//==================================================================================================
//								RJM Maszyny sp. z o.o.
//									13.05.2022
//
//	Obsługa przycisku niepodświetlanego
//	v1.0	|| TC v 3.1.4024.22		|| - pierwsza wersja
//==================================================================================================
INTERFACE I_Przycisk

//==================================================================================================
//								RJM Maszyny sp. z o.o.
//									13.05.2022
//
//	Sprawdzenie czy wciśnięty
//	v1.0	|| TC v 3.1.4024.22		|| - pierwsza wersja
//==================================================================================================
PROPERTY CzyNacisniety : Bool
GET
END_GET
END_PROPERTY

//==================================================================================================
//								RJM Maszyny sp. z o.o.
//									13.05.2022
//
//	Sprawdzenie czy puszczony
//	v1.0	|| TC v 3.1.4024.22		|| - pierwsza wersja
//==================================================================================================
PROPERTY CzyPuszczony : BOOL
GET
END_GET
END_PROPERTY

END_INTERFACE

(* stored: Version 1.1.0.1, ProductVersion 3.1.4024.11
   Itf I_Przycisk: Id {2cb2c177-f114-4664-a94f-2bdebc0b9573}
   Property CzyNacisniety: Id {53468298-c628-4961-8637-485b53b4fd24}
   Get Get: Id {2b1b4c90-fd99-447d-871d-48df7e65ead5}
   Property CzyPuszczony: Id {74b692fc-d4f4-49d4-85fa-76e663bc40c0}
   Get Get: Id {cd85e897-bb23-4b79-8e18-cc07778caa9d} *)
